TYPE sToken :
STRUCT
	boTokenRequest: BOOL;
	boTokenRelease: BOOL;
END_STRUCT
END_TYPE

(* stored: Version 1.1.0.1, ProductVersion 3.1.4026.13
   DUT sToken: Id {0859bd7f-0056-4eec-9a69-2b0f44b2bb78} *)
